FUNCTION_BLOCK SUB_DINT (* IEC 61131-3 DINT Subtraction *)
  (* Standard: 61131-3 *)
  (* Version 0.0, 2004-12-15, JHC, Rockwell Automation, Converted from SRC format. *)
  (* Compiler header: package fb.rt.plc.math; *)
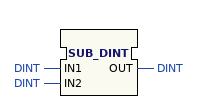
  VAR_INPUT
    IN1 : DINT; (* Minuend *)
    IN2 : DINT; (* Subtrahend *)
  END_VAR
  VAR_OUTPUT
    OUT : DINT; (* Difference *)
  END_VAR
END_FUNCTION_BLOCK
